FUNCTION_BLOCK FB_Remover EXTENDS FB_Conveyor
VAR_INPUT
    // Part is at conveyor entry
    bPartAtEntry: BOOL;
    // Part is at conveyor exit
    bPartAtExit: BOOL;
END_VAR
VAR_OUTPUT
    // Module is ready to receive part
    bReadyToReceivePart: BOOL;
    bPartProcessed: BOOL;
END_VAR
VAR
    // Part moving timeout
    fbMovingTimeout: TON;
    fbPartAtEntry: R_TRIG();
    nPartsOnConveyor: INT;
    // Current state of distributor
    eStateRemover: (R_IDLE, R_MOVE_PART, R_TRANSFER_TO_FOLLOWER, R_EMPTY_CONVEYOR, R_LOCKOUT);
END_VAR

SUPER^();
fbMovingTimeout();
fbPartAtEntry(CLK := bPartAtEntry);

IF fbPartAtEntry.Q THEN
    nPartsOnConveyor := nPartsOnConveyor + 1;
END_IF

CASE eStateRemover OF
    R_IDLE:
        SUPER^.Stop(bRunOut := TRUE);
        bReadyToReceivePart := TRUE;
        IF nPartsOnConveyor > 0 THEN
            eStateRemover := R_MOVE_PART;
        END_IF

    R_MOVE_PART:
        SUPER^.Start();
        fbMovingTimeout.IN := TRUE;
        IF PartAtExit() THEN
            fbMovingTimeout.IN := FALSE;
        ELSIF fbMovingTimeout.Q THEN
            // Throw error message: Part moving timeout
            fbMovingTimeout.IN := FALSE;
            nPartsOnConveyor := 0;
            eStateRemover := R_IDLE;
        END_IF

    R_TRANSFER_TO_FOLLOWER:
        SUPER^.Start();
        fbMovingTimeout.IN := TRUE;
        IF NOT bPartAtExit THEN
            fbMovingTimeout.IN := FALSE;
            nPartsOnConveyor := nPartsOnConveyor - 1;
            IF nPartsOnConveyor > 0 THEN
                eStateRemover := R_MOVE_PART;
            ELSE
                nPartsOnConveyor := 0;
                eStateRemover := R_IDLE;
            END_IF
        END_IF
        IF fbMovingTimeout.Q THEN
            // Throw error message: Part transfer moving timeout
            fbMovingTimeout.IN := FALSE;
            nPartsOnConveyor := 0;
            eStateRemover := R_IDLE;
        END_IF
END_CASE

// Return TRUE if part reach conveyor exit and state machine will go to next step
METHOD PRIVATE PartAtExit: BOOL
VAR_INPUT
END_VAR
IF bPartAtExit THEN
    eStateRemover := R_TRANSFER_TO_FOLLOWER;
ELSE
    PartAtExit := FALSE;
    RETURN;
END_IF

PartAtExit := TRUE;
END_METHOD

// Maximum duration for part to reach exit of conveyor
{attribute 'monitoring' := 'call'}
PROPERTY PUBLIC tMovingTimeout : TIME
GET
tMovingTimeout := fbMovingTimeout.PT;
END_GET
SET
fbMovingTimeout.PT := tMovingTimeout;
END_SET
END_PROPERTY

END_FUNCTION_BLOCK

(* stored: Version 1.1.0.1
   POU FB_Remover: Id {0bc5e74d-e01a-4eac-8057-39627e6c4303}, SpecialFunc None
   Method PartAtExit: Id {819b3435-f3e7-4c82-a928-abcde45f2cf7}
   Property tMovingTimeout: Id {2efb2728-9f0d-43d3-862b-fd68db65250b}
   Get Get: Id {36db0884-f442-4f2e-9856-af33307f7eb1}
   Set Set: Id {1a320144-ae0f-4a01-baec-2e883f795487} *)
